(* IEC 61131-3 sources: learning-path/05_oop_in_st/exercises/0_basic_valve_class/src, 3 files *)

(* ---- Tank.st ---- *)
NAMESPACE FluidHandling
    FUNCTION_BLOCK Tank
        VAR_INPUT
            cmdFill: BOOL;
            cmdEmpty: BOOL;
        END_VAR
        VAR_OUTPUT
            inletOpen: BOOL;
            outletOpen: BOOL;
        END_VAR
        VAR
            inlet: Valve;
            outlet: Valve;
        END_VAR

        inlet(cmdOpen := cmdFill,
                cmdClose:= NOT cmdFill,
                ctrlOpen => inletOpen);
        outlet(cmdOpen := cmdEmpty,
                cmdClose := NOT cmdEmpty,
                ctrlOpen => outletOpen);
    END_FUNCTION_BLOCK

END_NAMESPACE

(* ---- TankBase.st ---- *)
//Use the same namespace than the TYPE for the Valves state

NAMESPACE FluidHandlingClass

    CLASS TankBase
        VAR

        END_VAR

        METHOD PUBLIC Fill
            ;
        END_METHOD

        METHOD PUBLIC Flush
            ;
        END_METHOD

        METHOD PUBLIC Close
            ;
        END_METHOD

        METHOD PUBLIC Emptying
            ;
        END_METHOD

    END_CLASS

END_NAMESPACE

(* ---- basicValve.st ---- *)
//Use the same namespace than the TYPE for the Valves state

NAMESPACE FluidHandlingClass

    //HERE TYPE THE SOLUTION FOR THE CLASS VALVE

    END_NAMESPACE
